Staubli VAL3: onF5Event.pgx

program onF5Event()
  local num l_nSize
begin
  // look if the bButton is enable
  if bButton[4]
    //
    //  select it
    //
    call selectItem(nIndex)
    call trajType:getSizeItem(false,l_nSize)
    // go down
    if nIndex<l_nSize-1
      nSelect=nIndex+1
    endIf
    call buildList()
  endIf
end
